PROGRAM MAIN
VAR
END_VAR

END_PROGRAM

(* stored: Version 1.1.0.1
   POU MAIN: Id {119d41c0-ac57-4016-9f6f-39edac63d55a} *)
